INTERFACE ITF_MCMachineConfigure

METHOD PUBLIC AddConfiguration : BOOL
VAR_INPUT
	fbConfigure		: ITF_MCConfiguration;
END_VAR
END_METHOD

METHOD PUBLIC Configure : BOOL
VAR_INPUT
	fbMachineControl			: ITF_MCMachineControlConfigure;
END_VAR
END_METHOD

END_INTERFACE

(* stored: Version 1.1.0.1
   Itf ITF_MCMachineConfigure: Id {514aa852-a920-4435-b466-9727d5d56d90}
   Method AddConfiguration: Id {8cb64e8b-644a-4bc5-9fca-d874591a1392}
   Method Configure: Id {51f0da89-ace3-4acc-8f57-5a7a80c356a7} *)
